// TIA Portal V20 export
VAR_GLOBAL   // PLC tag table "F-IO"
   "BA010AZCRSP203.00" AT %I750.0 : Bool;   // BA010AD1 MODE SELECT AUTO : Main OP   {ExternalVisible false}
   "BA010AZCRSP203.01" AT %I750.1 : Bool;   // BA010AD1 HOME PBL : Main OP (GREEN)   {ExternalVisible false}
   "BA010AZCRSP203.02" AT %I750.2 : Bool;   // BA010AD1 SAFETY RESET PBL : Main OP (BLUE)   {ExternalVisible false}
   "BA010AZCRSP203.03" AT %I750.3 : Bool;   // BA010AD1SCS MODE SELECT AUTO : Main OP   {ExternalVisible false}
   "BA010AZCRSP203.04" AT %I750.4 : Bool;   // BA010AD1 MODE SELECT MANUAL : Main OP   {ExternalVisible false}
   "BA010AZCRSP203.05" AT %I750.5 : Bool;   // BA010AD1 ENABLE PBL : Main OP (WHITE)   {ExternalVisible false}
   "BA010AZCRSP203.07" AT %I750.7 : Bool;   // BA010AD1SCS MODE SELECT DISABLE : Main OP   {ExternalVisible false}
   "BA010AZCRSP204.00" AT %I760.0 : Bool;   // BA010AD1EMO00: Main OP   {ExternalVisible false}
   "BA010AZCRSP204.01" AT %I760.1 : Bool;   // SPARE   {ExternalVisible false}
   "BA010AZCRSP204.02" AT %I760.2 : Bool;   // SPARE   {ExternalVisible false}
   "BA010AZCRSP204.03" AT %I760.3 : Bool;   // SPARE   {ExternalVisible false}
   "BA010AZCRSP204.04" AT %I760.4 : Bool;   // BA010AD1EMO00: Main OP   {ExternalVisible false}
   "BA010AZCRSP204.05" AT %I760.5 : Bool;   // SPARE   {ExternalVisible false}
   "BA010AZCRSP204.06" AT %I760.6 : Bool;   // SPARE   {ExternalVisible false}
   "BA010AZCRSP204.07" AT %I760.7 : Bool;   // SPARE   {ExternalVisible false}
   "BA010AZCRSP205.00" AT %Q770.0 : Bool;   // BA010AD1 PENDANT REQUIRED PL LAMP ON : Main OP (YELLOW)   {ExternalVisible false}
   "BA010AZCRSP205.01" AT %Q770.1 : Bool;   // SPARE   {ExternalVisible false}
   "BA010AZCRSP205.02" AT %Q770.2 : Bool;   // BA010AD1 HOME PBL LAMP ON : Main OP (GREEN)   {ExternalVisible false}
   "BA010AZCRSP205.03" AT %Q770.3 : Bool;   // SPARE   {ExternalVisible false}
   "BA010AZCRSP205.04" AT %Q770.4 : Bool;   // SPARE   {ExternalVisible false}
   "BA010AZCRSP205.05" AT %Q770.5 : Bool;   // SPARE   {ExternalVisible false}
   "BA010AZCRSP205.06" AT %Q770.6 : Bool;   // SPARE   {ExternalVisible false}
   "BA010AZCRSP205.07" AT %Q770.7 : Bool;   // BA010AD1 SCS MODE SELECT DISABLE PL LAMP ON : Main OP(GREEN)   {ExternalVisible false}
   "BA010AZCRSBK01.00" AT %I4000.0 : Bool;   // BA010AE41EMO1: Unwinder   {ExternalVisible false}
   "BA010AZCRSBK01.01" AT %I4000.1 : Bool;   // BA010AE42EMO2: Cutter   {ExternalVisible false}
   "BA010AZCRSBK01.02" AT %I4000.2 : Bool;   // BA010AE43EMO3: Magazine   {ExternalVisible false}
   "BA010AZCRSBK01.03" AT %I4000.3 : Bool;   // BA010AE44EMO4: Conveyor   {ExternalVisible false}
   "BA010AZCRSBK01.04" AT %I4000.4 : Bool;   // BA010AE41EMO1: Unwinder   {ExternalVisible false}
   "BA010AZCRSBK01.05" AT %I4000.5 : Bool;   // BA010AE42EMO2: Cutter   {ExternalVisible false}
   "BA010AZCRSBK01.06" AT %I4000.6 : Bool;   // BA010AE43EMO3: Magazine   {ExternalVisible false}
   "BA010AZCRSBK01.07" AT %I4000.7 : Bool;   // BA010AE44EMO4: Conveyor   {ExternalVisible false}
   "BA010AZCRSBK01.10" AT %Q4000.0 : Bool;   // SPARE   {ExternalVisible false}
   "BA010AZCRSBK01.11" AT %Q4000.1 : Bool;   // SPARE   {ExternalVisible false}
   "BA010AZCRSBK01.12" AT %Q4000.2 : Bool;   // SPARE   {ExternalVisible false}
   "BA010AZCRSBK02.00" AT %I4010.0 : Bool;   // BA010AE1 SCS BOX SS.SETUP   {ExternalVisible false}
   "BA010AZCRSBK02.01" AT %I4010.1 : Bool;   // BA010AE1 SCS BOX SS.DISABLE   {ExternalVisible false}
   "BA010AZCRSBK02.02" AT %I4010.2 : Bool;   // PRX211 FRAME COVER SAFETY SENSOR   {ExternalVisible false}
   "BA010AZCRSBK02.03" AT %I4010.3 : Bool;   // SAFETY DOOR LOCK7.INPUT   {ExternalVisible false}
   "BA010AZCRSBK02.04" AT %I4010.4 : Bool;   // BA010AE1 SCS BOX SS.AUTO   {ExternalVisible false}
   "BA010AZCRSBK02.05" AT %I4010.5 : Bool;   // SPARE   {ExternalVisible false}
   "BA010AZCRSBK02.06" AT %I4010.6 : Bool;   // SPARE   {ExternalVisible false}
   "BA010AZCRSBK02.07" AT %I4010.7 : Bool;   // SAFETY DOOR LOCK7.INPUT   {ExternalVisible false}
   "BA010AZCRSBK02.10" AT %Q4010.0 : Bool;   // SCS box: Pendant required on, yellow   {ExternalVisible false}
   "BA010AZCRSBK02.11" AT %Q4010.1 : Bool;   // SCS box: SCS Disable mode selected, green   {ExternalVisible false}
   "BA010AZCRSBK02.12" AT %Q4010.2 : Bool;   // SAFETY DOOR LOCK7.OUTPUT   {ExternalVisible false}
   "BA010AZCRSBK03.00" AT %I4020.0 : Bool;   // BA010AE11 SS.AUTO LH ROLL CHANGE   {ExternalVisible false}
   "BA010AZCRSBK03.01" AT %I4020.1 : Bool;   // BA010AE12 SS.AUTO RH ROLL CHANGE   {ExternalVisible false}
   "BA010AZCRSBK03.02" AT %I4020.2 : Bool;   // PRX201 CART DETECT SENSOR1   {ExternalVisible false}
   "BA010AZCRSBK03.03" AT %I4020.3 : Bool;   // PRX202 CART DETECT SENSOR2   {ExternalVisible false}
   "BA010AZCRSBK03.04" AT %I4020.4 : Bool;   // BA010AE11 SS.CHANGE LH ROLL CHANGE   {ExternalVisible false}
   "BA010AZCRSBK03.05" AT %I4020.5 : Bool;   // BA010AE12 SS.CHANGE RH ROLL CHANGE   {ExternalVisible false}
   "BA010AZCRSBK03.06" AT %I4020.6 : Bool;   // PRX201 CART DETECT SENSOR1   {ExternalVisible false}
   "BA010AZCRSBK03.07" AT %I4020.7 : Bool;   // PRX202 CART DETECT SENSOR2   {ExternalVisible false}
   "BA010AZCRSBK03.10" AT %Q4020.0 : Bool;   // BA010AE11 IN PROGRESS LH ROLL CHANGE   {ExternalVisible false}
   "BA010AZCRSBK03.11" AT %Q4020.1 : Bool;   // BA010AE12 IN PROGRESS RH ROLL CHANGE   {ExternalVisible false}
   "BA010AZCRSBK03.12" AT %Q4020.2 : Bool;   // SPARE   {ExternalVisible false}
   "BA010AZCRSBK04.00" AT %I4030.0 : Bool;   // Gate EC TOP: Lock   {ExternalVisible false}
   "BA010AZCRSBK04.01" AT %I4030.1 : Bool;   // Gate EC TOP: Reset   {ExternalVisible false}
   "BA010AZCRSBK04.02" AT %I4030.2 : Bool;   // DIFFERENTIAL PRESSURE SWITCH 1 NC   {ExternalVisible false}
   "BA010AZCRSBK04.03" AT %I4030.3 : Bool;   // DIFFERENTIAL PRESSURE SWITCH 2 NC(Del)_7/29   {ExternalVisible false}
   "BA010AZCRSBK04.04" AT %I4030.4 : Bool;   // Gate EC.Top UnLock   {ExternalVisible false}
   "BA010AZCRSBK04.05" AT %I4030.5 : Bool;   // SPARE   {ExternalVisible false}
   "BA010AZCRSBK04.06" AT %I4030.6 : Bool;   // RESERVED   {ExternalVisible false}
   "BA010AZCRSBK04.07" AT %I4030.7 : Bool;   // RESERVED   {ExternalVisible false}
   "BA010AZCRSBK04.10" AT %Q4030.0 : Bool;   // Gate EC TOP: Lock lamp on   {ExternalVisible false}
   "BA010AZCRSBK04.11" AT %Q4030.1 : Bool;   // Gate EC TOP: Unlock lamp on   {ExternalVisible false}
   "BA010AZCRSBK04.12" AT %Q4030.2 : Bool;   // Gate EC TOP: Reset lamp on   {ExternalVisible false}
   "BA010AZCRSBK05.00" AT %I4040.0 : Bool;   // Gate EC.LH: Lock   {ExternalVisible false}
   "BA010AZCRSBK05.01" AT %I4040.1 : Bool;   // Gate EC.LH: Reset   {ExternalVisible false}
   "BA010AZCRSBK05.02" AT %I4040.2 : Bool;   // SPARE   {ExternalVisible false}
   "BA010AZCRSBK05.03" AT %I4040.3 : Bool;   // SPARE   {ExternalVisible false}
   "BA010AZCRSBK05.04" AT %I4040.4 : Bool;   // Gate EC LH: Unlock   {ExternalVisible false}
   "BA010AZCRSBK05.05" AT %I4040.5 : Bool;   // SPARE   {ExternalVisible false}
   "BA010AZCRSBK05.06" AT %I4040.6 : Bool;   // SPARE   {ExternalVisible false}
   "BA010AZCRSBK05.07" AT %I4040.7 : Bool;   // SPARE   {ExternalVisible false}
   "BA010AZCRSBK05.10" AT %Q4040.0 : Bool;   // Gate EC LH: Lock lamp on   {ExternalVisible false}
   "BA010AZCRSBK05.11" AT %Q4040.1 : Bool;   // Gate EC LH: Unlock lamp on   {ExternalVisible false}
   "BA010AZCRSBK05.12" AT %Q4040.2 : Bool;   // Gate EC LH: Reset lamp on   {ExternalVisible false}
   "BA010AZCRSBK06.00" AT %I4050.0 : Bool;   // BA010AZCRSDL1 UNWINDER MAIN DOOR   {ExternalVisible false}
   "BA010AZCRSBK06.01" AT %I4050.1 : Bool;   // BA010AZCRSDL2 UNWINDER LH DOOR   {ExternalVisible false}
   "BA010AZCRSBK06.02" AT %I4050.2 : Bool;   // BA010AZCRSDL3 UNWINDER RH DOOR   {ExternalVisible false}
   "BA010AZCRSBK06.03" AT %I4050.3 : Bool;   // SPARE   {ExternalVisible false}
   "BA010AZCRSBK06.04" AT %I4050.4 : Bool;   // BA010AZCRSDL1 UNWINDER MAIN DOOR   {ExternalVisible false}
   "BA010AZCRSBK06.05" AT %I4050.5 : Bool;   // BA010AZCRSDL2 UNWINDER LH DOOR   {ExternalVisible false}
   "BA010AZCRSBK06.06" AT %I4050.6 : Bool;   // BA010AZCRSDL3 UNWINDER RH DOOR   {ExternalVisible false}
   "BA010AZCRSBK06.07" AT %I4050.7 : Bool;   // SPARE   {ExternalVisible false}
   "BA010AZCRSBK06.10" AT %Q4050.0 : Bool;   // Gate EC.Top UnLock   {ExternalVisible false}
   "BA010AZCRSBK06.11" AT %Q4050.1 : Bool;   // Gate EC LH: Unlock   {ExternalVisible false}
   "BA010AZCRSBK06.12" AT %Q4050.2 : Bool;   // Gate EC RH: Unlock   {ExternalVisible false}
   "BA010AZCRSBK07.00" AT %I4060.0 : Bool;   // BA010AZCRSDL4 CUTTING DOOR   {ExternalVisible false}
   "BA010AZCRSBK07.01" AT %I4060.1 : Bool;   // BA010AZCRSDL5 MAGAZINE DOOR   {ExternalVisible false}
   "BA010AZCRSBK07.02" AT %I4060.2 : Bool;   // BA010AZCRSDL6 CONVEYOR DOOR   {ExternalVisible false}
   "BA010AZCRSBK07.03" AT %I4060.3 : Bool;   // SPARE   {ExternalVisible false}
   "BA010AZCRSBK07.04" AT %I4060.4 : Bool;   // BA010AZCRSDL4 CUTTING DOOR   {ExternalVisible false}
   "BA010AZCRSBK07.05" AT %I4060.5 : Bool;   // BA010AZCRSDL5 MAGAZINE DOOR   {ExternalVisible false}
   "BA010AZCRSBK07.06" AT %I4060.6 : Bool;   // BA010AZCRSDL6 CONVEYOR DOOR   {ExternalVisible false}
   "BA010AZCRSBK07.07" AT %I4060.7 : Bool;   // SPARE   {ExternalVisible false}
   "BA010AZCRSBK07.10" AT %Q4060.0 : Bool;   // GateCutter Unlock   {ExternalVisible false}
   "BA010AZCRSBK07.11" AT %Q4060.1 : Bool;   // GateMagazine Unlock   {ExternalVisible false}
   "BA010AZCRSBK07.12" AT %Q4060.2 : Bool;   // GateConveyor Unlock   {ExternalVisible false}
   "BA010AZCRSBK08.00" AT %I4070.0 : Bool;   // Gate EC RH: Lock   {ExternalVisible false}
   "BA010AZCRSBK08.01" AT %I4070.1 : Bool;   // Gate EC RH: Reset   {ExternalVisible false}
   "BA010AZCRSBK08.02" AT %I4070.2 : Bool;   // SPARE   {ExternalVisible false}
   "BA010AZCRSBK08.03" AT %I4070.3 : Bool;   // SPARE   {ExternalVisible false}
   "BA010AZCRSBK08.04" AT %I4070.4 : Bool;   // Gate EC RH: Unlock   {ExternalVisible false}
   "BA010AZCRSBK08.05" AT %I4070.5 : Bool;   // SPARE   {ExternalVisible false}
   "BA010AZCRSBK08.06" AT %I4070.6 : Bool;   // SPARE   {ExternalVisible false}
   "BA010AZCRSBK08.10" AT %Q4070.0 : Bool;   // Gate EC RH: Lock lamp on   {ExternalVisible false}
   "BA010AZCRSBK08.11" AT %Q4070.1 : Bool;   // Gate EC RH: Unlock lamp on   {ExternalVisible false}
   "BA010AZCRSBK08.12" AT %Q4070.2 : Bool;   // Gate EC RH: Reset lamp on   {ExternalVisible false}
   "BA010AZCRSBK09.00" AT %I4080.0 : Bool;   // Gate ScrapBox: Lock   {ExternalVisible false}
   "BA010AZCRSBK09.01" AT %I4080.1 : Bool;   // Gate ScrapBox : Reset   {ExternalVisible false}
   "BA010AZCRSBK09.02" AT %I4080.2 : Bool;   // SPARE   {ExternalVisible false}
   "BA010AZCRSBK09.03" AT %I4080.3 : Bool;   // SPARE   {ExternalVisible false}
   "BA010AZCRSBK09.04" AT %I4080.4 : Bool;   // Gate ScrapBox : Unlock   {ExternalVisible false}
   "BA010AZCRSBK09.05" AT %I4080.5 : Bool;   // SPARE   {ExternalVisible false}
   "BA010AZCRSBK09.06" AT %I4080.6 : Bool;   // SPARE   {ExternalVisible false}
   "BA010AZCRSBK09.07" AT %I4080.7 : Bool;   // SPARE   {ExternalVisible false}
   "BA010AZCRSBK09.10" AT %Q4080.0 : Bool;   // Gate ScrapBox : Lock lamp on   {ExternalVisible false}
   "BA010AZCRSBK09.11" AT %Q4080.1 : Bool;   // Gate ScrapBox : Unlock lamp on   {ExternalVisible false}
   "BA010AZCRSBK09.12" AT %Q4080.2 : Bool;   // Gate ScrapBox : Reset lamp on   {ExternalVisible false}
   "BA010AZCRMP105.00" AT %I150.0 : Bool;   // BA010AC1 MANIFOLD1 SOL POWER MC FEEDBACK   {ExternalVisible false}
   "BA010AZCRMP105.01" AT %I150.1 : Bool;   // SPARE   {ExternalVisible false}
   "BA010AZCRMP105.02" AT %I150.2 : Bool;   // SPARE   {ExternalVisible false}
   "BA010AZCRMP105.03" AT %I150.3 : Bool;   // SPARE   {ExternalVisible false}
   "BA010AZCRMP105.04" AT %I150.4 : Bool;   // BA010AC1 FFU POWER MC 1 FEEDBACK   {ExternalVisible false}
   "BA010AZCRMP105.05" AT %I150.5 : Bool;   // BA010AC1 FFU POWER MC 2 FEEDBACK   {ExternalVisible false}
   "BA010AZCRMP105.06" AT %I150.6 : Bool;   // SPARE   {ExternalVisible false}
   "BA010AZCRMP105.07" AT %I150.7 : Bool;   // SPARE   {ExternalVisible false}
   "BA010AZCRMP105.10" AT %I151.0 : Bool;   // SPARE   {ExternalVisible false}
   "BA010AZCRMP105.11" AT %I151.1 : Bool;   // SPARE   {ExternalVisible false}
   "BA010AZCRMP105.12" AT %I151.2 : Bool;   // SPARE   {ExternalVisible false}
   "BA010AZCRMP105.13" AT %I151.3 : Bool;   // SPARE   {ExternalVisible false}
   "BA010AZCRMP105.14" AT %I151.4 : Bool;   // SPARE   {ExternalVisible false}
   "BA010AZCRMP105.15" AT %I151.5 : Bool;   // SPARE   {ExternalVisible false}
   "BA010AZCRMP105.16" AT %I151.6 : Bool;   // SPARE   {ExternalVisible false}
   "BA010AZCRMP105.17" AT %I151.7 : Bool;   // SPARE   {ExternalVisible false}
   "BA010AZCRMP106.00" AT %Q160.0 : Bool;   // MANIFOLD1 SOL POWER MC ON   {ExternalVisible false}
   "BA010AZCRMP106.01" AT %Q160.1 : Bool;   // SPARE   {ExternalVisible false}
   "BA010AZCRMP106.02" AT %Q160.2 : Bool;   // SPARE   {ExternalVisible false}
   "BA010AZCRMP106.03" AT %Q160.3 : Bool;   // SPARE   {ExternalVisible false}
   "BA010AZCRMP106.04" AT %Q160.4 : Bool;   // FFU POWER MC ON 1   {ExternalVisible false}
   "BA010AZCRMP106.05" AT %Q160.5 : Bool;   // FFU POWER MC ON 2   {ExternalVisible false}
   "BA010AZCRMP106.06" AT %Q160.6 : Bool;   // SPARE   {ExternalVisible false}
   "BA010AZCRMP106.07" AT %Q160.7 : Bool;   // SPARE   {ExternalVisible false}
   "BA010AZCRFDI1.16" AT %I152.0 : Bool;   // Value state of MANIFOLD-1 SOL POWER MC FEEDBACK   {ExternalVisible false}
   "BA010AZCRFDI1.17" AT %I152.1 : Bool;   // Value state of SPARE   {ExternalVisible false}
   "BA010AZCRFDI1.20" AT %I152.4 : Bool;   // Value state of FFU POWER MC 1 FEEDBACK   {ExternalVisible false}
   "BA010AZCRFDI1.21" AT %I152.5 : Bool;   // Value state of FFU POWER MC 2 FEEDBACK   {ExternalVisible false}
   "BA010AZCRSBK08.07" AT %I4070.7 : Bool;   // SPARE   {ExternalVisible false}
   "BA010AZCRSP508.00" AT %I3500.0 : Bool;   // BA010AJ1PHMI EMO05: PHMI01   {ExternalVisible false}
   "BA010AZCRSP508.01" AT %I3500.1 : Bool;   // BA010AJ1PHMI ENABLE SWITCH: PHMI01   {ExternalVisible false}
   "BA010AZCRSP508.02" AT %I3500.2 : Bool;   // BA010AJ1PHMI EMO06: PHMI02   {ExternalVisible false}
   "BA010AZCRSP508.03" AT %I3500.3 : Bool;   // BA010AJ1PHMI ENABLE SWITCH: PHMI02   {ExternalVisible false}
   "BA010AZCRSP508.04" AT %I3500.4 : Bool;   // BA010AJ1PHMI EMO05: PHMI01   {ExternalVisible false}
   "BA010AZCRSP508.05" AT %I3500.5 : Bool;   // BA010AJ1PHMI ENABLE SWITCH: PHMI01   {ExternalVisible false}
   "BA010AZCRSP508.06" AT %I3500.6 : Bool;   // BA010AJ1PHMI EMO06: PHMI02   {ExternalVisible false}
   "BA010AZCRSP508.07" AT %I3500.7 : Bool;   // BA010AJ1PHMI ENABLE SWITCH: PHMI02   {ExternalVisible false}
   "BA010AZCRSP509.00" AT %Q3510.0 : Bool;   // BA010AJ1 UNWINDER EPC01 INTERLOCK   {ExternalVisible false}
   "BA010AZCRSP509.01" AT %Q3510.1 : Bool;   // BA010AJ1 UNWINDER EPC02 INTERLOCK   {ExternalVisible false}
   "BA010AZCRSP509.02" AT %Q3510.2 : Bool;   // BA010AJ1 UNWINDER EPC03 INTERLOCK   {ExternalVisible false}
   "BA010AZCRSP509.03" AT %Q3510.3 : Bool;   // SPARE   {ExternalVisible false}
   "BA010AZCRSP509.04" AT %Q3510.4 : Bool;   // SPARE   {ExternalVisible false}
   "BA010AZCRSP509.05" AT %Q3510.5 : Bool;   // SPARE   {ExternalVisible false}
   "BA010AZCRSP509.06" AT %Q3510.6 : Bool;   // SPARE   {ExternalVisible false}
   "BA010AZCRSP509.07" AT %Q3510.7 : Bool;   // SPARE   {ExternalVisible false}
   BA010AZCRPM01 AT %Q2500.0 : Bool;   // BA010AZCRPM01 MANIFOLD SAFE POWER   {ExternalVisible false}
   BA010AZCRPM02 AT %Q2505.0 : Bool;   // BA010AZCRPM02 MANIFOLD SAFE POWER   {ExternalVisible false}
   BA010AZCRPM03 AT %Q2510.0 : Bool;   // BA010AZCRPM03 MANIFOLD SAFE POWER   {ExternalVisible false}
   BA010AZCRPM04 AT %Q2515.0 : Bool;   // BA010AZCRPM04 MANIFOLD SAFE POWER   {ExternalVisible false}
   "BA010AZCRSP203.06" AT %I750.6 : Bool;   // BA010AD1SCS MODE SELECT SETUP : Main OP   {ExternalVisible false}
   BA010AZCRPM05 AT %Q2520.0 : Bool;   // BA010AZCRPM05 MANIFOLD SAFE POWER   {ExternalVisible false}
   BA010AZCRPM06 AT %Q2525.0 : Bool;   // BA010AZCRPM06 MANIFOLD SAFE POWER   {ExternalVisible false}
   "BA010AZCRSP513.00" AT %IW3118 : Int;   // LEFT UNWINDER RADIUS SENSOR   {ExternalVisible false}
   "BA010AZCRSP513.01" AT %IW3120 : Int;   // RIGHT UNWINDER RADIUS SENSOR   {ExternalVisible false}
   "BA010AZCRSP513.02" AT %IW3122 : Int;   // SPARE   {ExternalVisible false}
   "BA010AZCRSP513.03" AT %IW3124 : Int;   // SPARE   {ExternalVisible false}
END_VAR
